TYPE STCcdData_1 :
STRUCT
	iorder:DINT;  //功能码  2  3   4    
	strCode:STRING   ;//二维码
	strShortData: STRING; //短路测试数据 128
	strBetryName: STRING;//文件名
	strHotPress: STRING;//热压参数
END_STRUCT
END_TYPE

(* stored: Version 1.1.0.1, ProductVersion 3.1.4024.9
   DUT STCcdData_1: Id {ce9d6b4d-f334-42db-9d0b-afcf27b3d9c3} *)
